// TIA Portal V18 export
DATA_BLOCK "MC_Power_DB"   // DB13
// stored: AutoNumber true, DBAccessibleFromOPCUA true, InstanceOfName MC_Power, OfSystemLibElement MC_Power, OfSystemLibVersion 7.0
"MC_Power"
   // VAR_INPUT
   //    Axis : TO_Axis;
   //    Enable : Bool;
   //    StartMode : Int;
   //    StopMode : Int;
   // END_VAR
   // VAR_OUTPUT
   //    Status : Bool;
   //    Busy : Bool;
   //    Error : Bool;
   //    ErrorID : Word;
   //    ErrorInfo : Word;
   // END_VAR
   // VAR
   //    FB_ID : DInt;
   // END_VAR
BEGIN
END_DATA_BLOCK
